// TIA Portal V16 export
// export: Created 2022-03-28T07:44:07.8293901Z, ExportSetting WithDefaults, DisplayName Totally Integrated Automation Portal, DisplayVersion V16 Update 5, DisplayName TIA Portal Version Control Interface, DisplayVersion V16 Update 2, DisplayName TIA Portal Openness, DisplayVersion V16 Update 5, DisplayName STEP 7 Professional, DisplayVersion V16 Update 5, DisplayName STEP 7 Safety, DisplayVersion V16, DisplayName WinCC Professional, DisplayVersion V16 Update 5
DATA_BLOCK "db_Programs"   // DB101
{ S7_Optimized_Access := 'TRUE' }
VERSION : 0.1
// stored: AutoNumber false, IsOnlyStoredInLoadMemory false, IsRetainMemResEnabled false, IsWriteProtectedInAS false, MemoryReserve 100
   VAR RETAIN
      diProgramSelection : DInt := 8;
   END_VAR
   VAR
      bSaveKey : Bool := FALSE;
      diStepCounter : DInt := 1;
      strShortBolt : String[16] := '';
      strMediumBolt : String[16] := '';
      strLongBolt : String[16] := '';
      strSmallNut : String[16] := '';
      strBigNut : String[16] := '';
   END_VAR
   VAR RETAIN
      udtProgram { S7_SetPoint := 'True'} : Array[1..10] of "udtProgram";
      udtWorkProgram { S7_SetPoint := 'True'} : "udtProgram";
   END_VAR
   VAR
      udtWorkStep { S7_SetPoint := 'True'} : "udtStep";
   END_VAR
BEGIN
   udtProgram[1].strName := 'TCS327=178';
   udtProgram[2].strName := 'TCS327=193';
   udtProgram[3].strName := 'TCS327=192';
   udtProgram[4].strName := 'TCS327=181';
   udtProgram[5].strName := 'TCS327=186';
   udtProgram[6].strName := 'TCS327=200';
   udtProgram[7].strName := 'TCS327=188';
   udtProgram[8].strName := 'TCS327=190';
   udtProgram[9].strName := 'TCS327=197';
   udtProgram[10].strName := '191.33476980';
   udtProgram[1].udtStep[1..4].iAction := 2;
   udtProgram[1].udtStep[5..7].iAction := 1;
   udtProgram[1].udtStep[8..10].iAction := 0;
   udtProgram[2].udtStep[1].iAction := 6;
   udtProgram[2].udtStep[2].iAction := 5;
   udtProgram[2].udtStep[3..4].iAction := 3;
   udtProgram[2].udtStep[5..10].iAction := 0;
   udtProgram[3].udtStep[1..2].iAction := 1;
   udtProgram[3].udtStep[3..10].iAction := 0;
   udtProgram[4].udtStep[1..3].iAction := 6;
   udtProgram[4].udtStep[4].iAction := 1;
   udtProgram[4].udtStep[5..10].iAction := 0;
   udtProgram[5].udtStep[1..2].iAction := 2;
   udtProgram[5].udtStep[3..10].iAction := 0;
   udtProgram[6].udtStep[1].iAction := 5;
   udtProgram[6].udtStep[2].iAction := 1;
   udtProgram[6].udtStep[3..10].iAction := 0;
   udtProgram[7].udtStep[1].iAction := 5;
   udtProgram[7].udtStep[2].iAction := 1;
   udtProgram[7].udtStep[3..10].iAction := 0;
   udtProgram[8].udtStep[1].iAction := 6;
   udtProgram[8].udtStep[2].iAction := 4;
   udtProgram[8].udtStep[3..7].iAction := 1;
   udtProgram[8].udtStep[8..10].iAction := 0;
   udtProgram[9].udtStep[1..3].iAction := 4;
   udtProgram[9].udtStep[4..10].iAction := 0;
   udtProgram[10].udtStep[1..10].iAction := 0;
   udtProgram[1].udtStep[1..7].iPG := 3;
   udtProgram[1].udtStep[8..10].iPG := 0;
   udtProgram[2].udtStep[1].iPG := 22;
   udtProgram[2].udtStep[2].iPG := 23;
   udtProgram[2].udtStep[3..4].iPG := 3;
   udtProgram[2].udtStep[5].iPG := 9;
   udtProgram[2].udtStep[6..7].iPG := 1;
   udtProgram[2].udtStep[8..10].iPG := 0;
   udtProgram[3].udtStep[1..2].iPG := 3;
   udtProgram[3].udtStep[3..10].iPG := 0;
   udtProgram[4].udtStep[1..3].iPG := 22;
   udtProgram[4].udtStep[4].iPG := 3;
   udtProgram[4].udtStep[5..10].iPG := 0;
   udtProgram[5].udtStep[1..3].iPG := 3;
   udtProgram[5].udtStep[4..10].iPG := 0;
   udtProgram[6].udtStep[1].iPG := 5;
   udtProgram[6].udtStep[2].iPG := 3;
   udtProgram[6].udtStep[3..10].iPG := 0;
   udtProgram[7].udtStep[1].iPG := 5;
   udtProgram[7].udtStep[2].iPG := 3;
   udtProgram[7].udtStep[3..10].iPG := 0;
   udtProgram[8].udtStep[1].iPG := 1;
   udtProgram[8].udtStep[2].iPG := 2;
   udtProgram[8].udtStep[3..7].iPG := 3;
   udtProgram[8].udtStep[8..10].iPG := 0;
   udtProgram[9].udtStep[1..3].iPG := 1;
   udtProgram[9].udtStep[4..10].iPG := 0;
   udtProgram[10].udtStep[1..10].iPG := 0;
   udtProgram[1].udtStep[1].iLamp := 2;
   udtProgram[1].udtStep[2].iLamp := 1;
   udtProgram[1].udtStep[3].iLamp := 3;
   udtProgram[1].udtStep[4].iLamp := 4;
   udtProgram[1].udtStep[5].iLamp := 5;
   udtProgram[1].udtStep[6].iLamp := 6;
   udtProgram[1].udtStep[7].iLamp := 7;
   udtProgram[1].udtStep[8..10].iLamp := 0;
   udtProgram[2].udtStep[1..2].iLamp := 2;
   udtProgram[2].udtStep[3].iLamp := 3;
   udtProgram[2].udtStep[4].iLamp := 4;
   udtProgram[2].udtStep[5].iLamp := 5;
   udtProgram[2].udtStep[6].iLamp := 6;
   udtProgram[2].udtStep[7].iLamp := 7;
   udtProgram[2].udtStep[8..10].iLamp := 0;
   udtProgram[3].udtStep[1].iLamp := 1;
   udtProgram[3].udtStep[2].iLamp := 2;
   udtProgram[3].udtStep[3..10].iLamp := 0;
   udtProgram[4].udtStep[1].iLamp := 1;
   udtProgram[4].udtStep[2].iLamp := 2;
   udtProgram[4].udtStep[3].iLamp := 3;
   udtProgram[4].udtStep[4..10].iLamp := 0;
   udtProgram[5].udtStep[1].iLamp := 1;
   udtProgram[5].udtStep[2].iLamp := 2;
   udtProgram[5].udtStep[3].iLamp := 3;
   udtProgram[5].udtStep[4..10].iLamp := 0;
   udtProgram[6].udtStep[1].iLamp := 1;
   udtProgram[6].udtStep[2].iLamp := 2;
   udtProgram[6].udtStep[3..10].iLamp := 0;
   udtProgram[7].udtStep[1].iLamp := 1;
   udtProgram[7].udtStep[2].iLamp := 2;
   udtProgram[7].udtStep[3..10].iLamp := 0;
   udtProgram[8].udtStep[1].iLamp := 7;
   udtProgram[8].udtStep[2].iLamp := 1;
   udtProgram[8].udtStep[3].iLamp := 6;
   udtProgram[8].udtStep[4].iLamp := 5;
   udtProgram[8].udtStep[5].iLamp := 3;
   udtProgram[8].udtStep[6].iLamp := 2;
   udtProgram[8].udtStep[7].iLamp := 4;
   udtProgram[8].udtStep[8..10].iLamp := 0;
   udtProgram[9].udtStep[1].iLamp := 1;
   udtProgram[9].udtStep[2].iLamp := 2;
   udtProgram[9].udtStep[3].iLamp := 3;
   udtProgram[9].udtStep[4..10].iLamp := 0;
   udtProgram[10].udtStep[1..10].iLamp := 0;
   udtWorkProgram.strName := 'TCS327=190';
   udtWorkProgram.udtStep[1].iAction := 6;
   udtWorkProgram.udtStep[2].iAction := 4;
   udtWorkProgram.udtStep[3..7].iAction := 1;
   udtWorkProgram.udtStep[8..10].iAction := 0;
   udtWorkProgram.udtStep[1].iPG := 1;
   udtWorkProgram.udtStep[2].iPG := 2;
   udtWorkProgram.udtStep[3..7].iPG := 3;
   udtWorkProgram.udtStep[8..10].iPG := 0;
   udtWorkProgram.udtStep[1].iLamp := 7;
   udtWorkProgram.udtStep[2].iLamp := 1;
   udtWorkProgram.udtStep[3].iLamp := 6;
   udtWorkProgram.udtStep[4].iLamp := 5;
   udtWorkProgram.udtStep[5].iLamp := 3;
   udtWorkProgram.udtStep[6].iLamp := 2;
   udtWorkProgram.udtStep[7].iLamp := 4;
   udtWorkProgram.udtStep[8..10].iLamp := 0;
   udtWorkStep.iAction := 6;
   udtWorkStep.iPG := 1;
   udtWorkStep.iLamp := 7;
END_DATA_BLOCK
